(* CODESYS project Teste.project

Project tree, tasks and I/O mapping:
  Device : CODESYS Control Win V3, 3S - Smart Software Solutions GmbH, order no. 305021, version 3.5.11.40
    application Application
      libraries: Standard, * (System)
      task MainTask (cyclic, interval t#20ms, priority 1) calls Main
      program Main [ST]
      global variables Variaveis
      Carregamento/
        function UpdateAlarms [ST]
        function IniciarProcessoCarregamento [ST]
        function ExecutarCarregamento [ST]
        function ContinuarCarregamento [ST]
        function DesligarEquipamentosAposCarregamento [ST]
        function block ControleCarregamento [ST]
      ControleDescarregamento/
        function block ControleDescarregamento [ST]
        function UpdateAlarmsDescarregamento [ST]
        function IniciarProcessoDescarregamento [ST]
        function ExecutarDescarregamento [ST]
        function DesligarEquipamentosAposDescarregamento [ST]
      Geral/
        function VerificarCondicoesMudancaModo [ST]
      Symbols
*)

// Device/Application/Variaveis
VAR_GLOBAL
    // Variáveis de Comando
    CMD_INICIAR_CARREGAMENTO: BOOL := FALSE;
    CMD_INICIAR_DESCARREGAMENTO: BOOL := FALSE;

    // Variáveis do Caminhão
    CAMINHAO_POSICIONADO: BOOL := FALSE;
    CAPACIDADE_CAMINHAO: REAL := 0.0;

    // Variáveis dos Silos
    PESO_SILO1: REAL := 0.0;
    PESO_SILO2: REAL := 0.0;
    NIVEL_BAIXO_SILO1: BOOL := FALSE;
    NIVEL_BAIXO_SILO2: BOOL := FALSE;

    // Variáveis de Equipamentos
    VENTILACAO_SILO1: BOOL := FALSE;
    VENTILACAO_SILO2: BOOL := FALSE;
    ALIMENTADOR_MOEGA1_ON: BOOL := FALSE;
    ALIMENTADOR_MOEGA2_ON: BOOL := FALSE;
    TRANSPORTADOR_SAIDA_ON: BOOL := FALSE;
    MOEGA_PESAGEM_ON: BOOL := FALSE;
    TRANSPORTADOR_ENTRADA_ON: BOOL := FALSE;

    // Variáveis de Pesagem
    PESO_MOEGA: REAL := 0.0;
    TaxaTransferencia: REAL := 0.0;

    // Variáveis de Alarmes
    ALARME_CARREGAMENTO: BOOL := FALSE;
    ALARME_DESCARREGAMENTO: BOOL := FALSE;

    // Variáveis de Controle de Processo
    INICIAR_CARREGAMENTO: BOOL := FALSE;
    INICIAR_DESCARREGAMENTO: BOOL := FALSE;
    inicio_carregamento: TIME;
    inicio_descarregamento: TIME;
    SiloSelecionado: INT := 0;
	DESVIADOR_MANGUEIRA: INT;

    // Variáveis Adicionais
    VAGAO_POSICIONADO: BOOL := FALSE;
    CAPACIDADE_VAGAO: REAL := 1000.0; // Capacidade do vagão em kg

    // Modo de Operação: TRUE para Automático, FALSE para Manual
    Modo_Automatico_Carregamento: BOOL := FALSE; // FALSE = Manual, TRUE = Automático
    Modo_Automatico_Descarregamento: BOOL := FALSE; // FALSE = Manual, TRUE = Automático

    // Variáveis de Controle Manual
    CMD_MANUAL_VENTILACAO_SILO1: BOOL := FALSE;
    CMD_MANUAL_VENTILACAO_SILO2: BOOL := FALSE;
    CMD_MANUAL_ALIMENTADOR_MOEGA1_ON: BOOL := FALSE;
    CMD_MANUAL_ALIMENTADOR_MOEGA2_ON: BOOL := FALSE;
    CMD_MANUAL_TRANSPORTADOR_ENTRADA_ON: BOOL := FALSE;
    CMD_MANUAL_TRANSPORTADOR_SAIDA_ON: BOOL := FALSE;
    CMD_MANUAL_MOEGA_PESAGEM_ON: BOOL := FALSE;
    CMD_MANUAL_ALIMENTADOR_SAIDA_ON: BOOL := FALSE;

    // Condições de Equipamentos e Alarmes
    Equipamentos_Desligados: BOOL := TRUE;
    Alarmes_Ativos: BOOL := FALSE;
    Alarme_Nivel_Baixo_Ativo: BOOL := FALSE;
    Alarme_Nivel_Alto_Ativo: BOOL := FALSE;
END_VAR

// Device/Application/Main
PROGRAM Main
VAR_INPUT
    
    CMD_INICIAR_CARREGAMENTO: BOOL;
    CMD_INICIAR_DESCARREGAMENTO: BOOL;

    CAMINHAO_POSICIONADO: BOOL;
    CAPACIDADE_CAMINHAO: REAL;
    
    PESO_SILO1: REAL;
    PESO_SILO2: REAL;

    Modo_Automatico: BOOL; 

    CMD_MANUAL_VENTILACAO_SILO1: BOOL;
    CMD_MANUAL_VENTILACAO_SILO2: BOOL;
    CMD_MANUAL_ALIMENTADOR_MOEGA1_ON: BOOL;
    CMD_MANUAL_ALIMENTADOR_MOEGA2_ON: BOOL;
    CMD_MANUAL_TRANSPORTADOR_ENTRADA_ON: BOOL;
    CMD_MANUAL_TRANSPORTADOR_SAIDA_ON: BOOL;
    CMD_MANUAL_MOEGA_PESAGEM_ON: BOOL;
    CMD_MANUAL_ALIMENTADOR_SAIDA_ON: BOOL;
END_VAR

VAR_OUTPUT
    
    VENTILACAO_SILO1: BOOL;
    VENTILACAO_SILO2: BOOL;
    ALIMENTADOR_MOEGA1_ON: BOOL;
    ALIMENTADOR_MOEGA2_ON: BOOL;
    TRANSPORTADOR_SAIDA_ON: BOOL;
    MOEGA_PESAGEM_ON: BOOL;
    TRANSPORTADOR_ENTRADA_ON: BOOL;
    DESVIADOR_MANGUEIRA: INT;
END_VAR

VAR
    
    NIVEL_BAIXO_SILO1: BOOL;
    NIVEL_BAIXO_SILO2: BOOL;
    NIVEL_ALTO_SILO1: BOOL;
    NIVEL_ALTO_SILO2: BOOL;
    
    PESO_MOEGA: REAL;
    TaxaTransferenciaCarregamento: REAL := 50.0;
    TaxaTransferenciaDescarregamento: REAL := 100.0;
    
    ALARME_CARREGAMENTO: BOOL;
    ALARME_DESCARREGAMENTO: BOOL;
    
    INICIAR_CARREGAMENTO: BOOL;
    INICIAR_DESCARREGAMENTO: BOOL;
    inicio_carregamento: TIME;
    inicio_descarregamento: TIME;
    SiloSelecionado: INT;
    
    VAGAO_POSICIONADO: BOOL;
    CAPACIDADE_VAGAO: REAL := 1000.0;
    VAGAO_CAPACIDADE_RESTANTE: REAL := 0.0; 
    VAGAO_POSICIONADO_ANTERIOR: BOOL := FALSE;
    
    lastUpdateTime: TIME;
    elapsedTime: REAL;
    CAMINHAO_CHEIO: BOOL;
    equipmentOffTime: TIME;
    VAGAO_CHEIO: BOOL; 
END_VAR

//
// Update Alarms
//ALARME_CARREGAMENTO := NOT CAMINHAO_POSICIONADO OR (CAPACIDADE_CAMINHAO < 200 OR CAPACIDADE_CAMINHAO > 800);
//IF ALARME_CARREGAMENTO THEN
  //  INICIAR_CARREGAMENTO := FALSE;
//END_IF;

//ALARME_DESCARREGAMENTO := NOT VAGAO_POSICIONADO OR (PESO_SILO1 >= 2400 OR PESO_SILO2 >= 2400);
//IF ALARME_DESCARREGAMENTO THEN
  //  INICIAR_DESCARREGAMENTO := FALSE;
//END_IF;

IF PESO_SILO1 < 100 THEN
    NIVEL_BAIXO_SILO1 := TRUE;
ELSE
    NIVEL_BAIXO_SILO1 := FALSE;    
END_IF

IF PESO_SILO2 < 100 THEN
    NIVEL_BAIXO_SILO2 := TRUE;
ELSE
    NIVEL_BAIXO_SILO2 := FALSE;    
END_IF

IF PESO_SILO1 > 2400 THEN
	NIVEL_ALTO_SILO1 := TRUE;
ELSE
    NIVEL_ALTO_SILO1 := FALSE;	
END_IF

IF PESO_SILO2 > 2400 THEN
	NIVEL_ALTO_SILO2 := TRUE;
ELSE 
    NIVEL_ALTO_SILO2 := FALSE;	
END_IF

elapsedTime := TIME_TO_REAL(TIME() - lastUpdateTime) / 1000.0;
lastUpdateTime := TIME();

IF VAGAO_POSICIONADO AND NOT VAGAO_POSICIONADO_ANTERIOR THEN
    VAGAO_CAPACIDADE_RESTANTE := CAPACIDADE_VAGAO;
    VAGAO_POSICIONADO_ANTERIOR := TRUE;
	VAGAO_CHEIO := FALSE;
ELSIF NOT VAGAO_POSICIONADO THEN
    VAGAO_POSICIONADO_ANTERIOR := FALSE;
END_IF;


IF Modo_Automatico THEN
    
    IF NOT INICIAR_CARREGAMENTO AND CMD_INICIAR_CARREGAMENTO AND CAMINHAO_POSICIONADO AND ((PESO_SILO1 - 100) + (PESO_SILO2 - 100) >= CAPACIDADE_CAMINHAO) AND (CAPACIDADE_CAMINHAO >= 200 AND CAPACIDADE_CAMINHAO <= 800 AND (REAL_TO_INT(CAPACIDADE_CAMINHAO) MOD 50 = 0)) THEN
        INICIAR_CARREGAMENTO := TRUE;
        inicio_carregamento := TIME();
        ALARME_CARREGAMENTO := FALSE;

        
        IF PESO_SILO1 >= PESO_SILO2 THEN
            SiloSelecionado := 1;
            VENTILACAO_SILO1 := TRUE;
            ALIMENTADOR_MOEGA1_ON := TRUE;
            ALIMENTADOR_MOEGA2_ON := FALSE;
        ELSE
            SiloSelecionado := 2;
            VENTILACAO_SILO2 := TRUE;
            ALIMENTADOR_MOEGA2_ON := TRUE;
            ALIMENTADOR_MOEGA1_ON := FALSE;
        END_IF;
    END_IF;

    IF INICIAR_CARREGAMENTO THEN
        
        IF (PESO_SILO1 >= 100 OR PESO_SILO2 >= 100) THEN
            TRANSPORTADOR_SAIDA_ON := TRUE;
            MOEGA_PESAGEM_ON := TRUE;
           
            IF PESO_MOEGA <= CAPACIDADE_CAMINHAO  THEN
                PESO_MOEGA := PESO_MOEGA + TaxaTransferenciaCarregamento * elapsedTime;
                IF SiloSelecionado = 1 AND (NOT NIVEL_BAIXO_SILO1) THEN
                    PESO_SILO1 := PESO_SILO1 - TaxaTransferenciaCarregamento * elapsedTime;
					VENTILACAO_SILO1 := TRUE;
                    ALIMENTADOR_MOEGA1_ON := TRUE;
					VENTILACAO_SILO2 := FALSE;
                    ALIMENTADOR_MOEGA2_ON := FALSE;
                    IF NIVEL_BAIXO_SILO1 THEN
                        
                        SiloSelecionado := 2;
                        VENTILACAO_SILO1 := FALSE;
                        VENTILACAO_SILO2 := TRUE;
                        ALIMENTADOR_MOEGA1_ON := FALSE;
                        ALIMENTADOR_MOEGA2_ON := TRUE;
                    END_IF;
                ELSE
                    PESO_SILO2 := PESO_SILO2 - TaxaTransferenciaCarregamento * elapsedTime;
                    VENTILACAO_SILO2 := TRUE;
                    ALIMENTADOR_MOEGA2_ON := TRUE;
					VENTILACAO_SILO1 := FALSE;
                    ALIMENTADOR_MOEGA1_ON := FALSE;
                    IF NIVEL_BAIXO_SILO2 THEN
                        SiloSelecionado := 1;
                        VENTILACAO_SILO2 := FALSE;
                        VENTILACAO_SILO1 := TRUE;
                        ALIMENTADOR_MOEGA2_ON := FALSE;
                        ALIMENTADOR_MOEGA1_ON := TRUE;
                    END_IF;
                END_IF;
            END_IF
        ELSE
            ALARME_CARREGAMENTO := TRUE;
            INICIAR_CARREGAMENTO := FALSE;
        END_IF;

        IF PESO_MOEGA >= CAPACIDADE_CAMINHAO THEN
            CAMINHAO_CHEIO := TRUE;
            INICIAR_CARREGAMENTO := FALSE; 
            equipmentOffTime := TIME(); 
        END_IF;
    END_IF;

   
    IF CAMINHAO_CHEIO THEN
        IF (TIME() - equipmentOffTime >= T#1S) THEN
            MOEGA_PESAGEM_ON := FALSE;
        END_IF;
        IF (TIME() - equipmentOffTime >= T#2S) THEN
            TRANSPORTADOR_SAIDA_ON := FALSE;
        END_IF;
        IF (TIME() - equipmentOffTime >= T#3S) THEN
            ALIMENTADOR_MOEGA1_ON := FALSE;
            ALIMENTADOR_MOEGA2_ON := FALSE;
        END_IF;
        IF (TIME() - equipmentOffTime >= T#5S) THEN
            VENTILACAO_SILO1 := FALSE;
            VENTILACAO_SILO2 := FALSE;
            CAMINHAO_CHEIO := FALSE; 
        END_IF;
    END_IF;
	
    IF NOT INICIAR_DESCARREGAMENTO AND CMD_INICIAR_DESCARREGAMENTO AND VAGAO_POSICIONADO AND (PESO_SILO1 + PESO_SILO2 < 5000) AND (NOT VAGAO_CHEIO) AND NOT (NIVEL_ALTO_SILO1 AND NIVEL_ALTO_SILO2) THEN
        IF NOT ALARME_DESCARREGAMENTO THEN
            INICIAR_DESCARREGAMENTO := TRUE;
            inicio_descarregamento := TIME();
           
            IF (PESO_SILO1 <= PESO_SILO2) AND (NOT NIVEL_ALTO_SILO1) THEN
                //SiloSelecionado := 1;
                DESVIADOR_MANGUEIRA := 1;
                VENTILACAO_SILO1 := TRUE;
                VENTILACAO_SILO2 := FALSE;
            ELSE
               // SiloSelecionado := 2;
                DESVIADOR_MANGUEIRA := 2;
                VENTILACAO_SILO2 := TRUE;
                VENTILACAO_SILO1 := FALSE;
            END_IF;
        ELSE
            INICIAR_DESCARREGAMENTO := FALSE;
			ALARME_DESCARREGAMENTO  := TRUE;
        END_IF;
    END_IF;

    IF INICIAR_DESCARREGAMENTO THEN
        TRANSPORTADOR_ENTRADA_ON := TRUE;
        IF VAGAO_CAPACIDADE_RESTANTE > 0 THEN
            IF (NOT NIVEL_ALTO_SILO1) AND (DESVIADOR_MANGUEIRA = 1) THEN
                PESO_SILO1 := PESO_SILO1 + TaxaTransferenciaDescarregamento * elapsedTime;
                VAGAO_CAPACIDADE_RESTANTE := VAGAO_CAPACIDADE_RESTANTE - TaxaTransferenciaDescarregamento * elapsedTime;
				DESVIADOR_MANGUEIRA := 1;
				VENTILACAO_SILO1 := TRUE;
				VENTILACAO_SILO2 := FALSE;
                IF NIVEL_ALTO_SILO1 THEN
                    
                   //SiloSelecionado := 2;
                   DESVIADOR_MANGUEIRA := 2;
                   VENTILACAO_SILO1 := FALSE;
                   VENTILACAO_SILO2 := TRUE;
               END_IF;
            ELSE
                PESO_SILO2 := PESO_SILO2 + TaxaTransferenciaDescarregamento * elapsedTime;
                VAGAO_CAPACIDADE_RESTANTE := VAGAO_CAPACIDADE_RESTANTE - TaxaTransferenciaDescarregamento * elapsedTime;
				DESVIADOR_MANGUEIRA := 2;
				VENTILACAO_SILO2 := TRUE;
				VENTILACAO_SILO1 := FALSE;
                 IF NIVEL_ALTO_SILO2 THEN
                   
                   //SiloSelecionado := 1;
                   DESVIADOR_MANGUEIRA := 1;
                   VENTILACAO_SILO2 := FALSE;
                   VENTILACAO_SILO1 := TRUE;
                END_IF;
            END_IF;

            IF VAGAO_CAPACIDADE_RESTANTE <= 0 THEN
                VAGAO_CHEIO := TRUE;
                INICIAR_DESCARREGAMENTO := FALSE; 
                equipmentOffTime := TIME(); 
            END_IF;
        END_IF;
    END_IF;

    IF VAGAO_CHEIO THEN
        IF (TIME() - equipmentOffTime >= T#2S) THEN
            TRANSPORTADOR_ENTRADA_ON := FALSE;
        END_IF;
        IF (TIME() - equipmentOffTime >= T#5S) THEN
            IF DESVIADOR_MANGUEIRA = 1 THEN
                VENTILACAO_SILO1 := FALSE;
            ELSE
                VENTILACAO_SILO2 := FALSE;
            END_IF;
           // VAGAO_CHEIO := FALSE; 
        END_IF;
    END_IF;
END_IF


IF NOT Modo_Automatico THEN
    
    VENTILACAO_SILO1 := CMD_MANUAL_VENTILACAO_SILO1;
    VENTILACAO_SILO2 := CMD_MANUAL_VENTILACAO_SILO2;
    ALIMENTADOR_MOEGA1_ON := CMD_MANUAL_ALIMENTADOR_MOEGA1_ON;
    ALIMENTADOR_MOEGA2_ON := CMD_MANUAL_ALIMENTADOR_MOEGA2_ON;
    TRANSPORTADOR_SAIDA_ON := CMD_MANUAL_TRANSPORTADOR_SAIDA_ON;
    MOEGA_PESAGEM_ON := CMD_MANUAL_MOEGA_PESAGEM_ON;
    
    // Manual Unloading
    VENTILACAO_SILO1 := CMD_MANUAL_VENTILACAO_SILO1;
    VENTILACAO_SILO2 := CMD_MANUAL_VENTILACAO_SILO2;
    TRANSPORTADOR_ENTRADA_ON := CMD_MANUAL_TRANSPORTADOR_ENTRADA_ON;
END_IF;

END_PROGRAM

// Device/Application/Carregamento/UpdateAlarms
FUNCTION UpdateAlarms : BOOL
VAR_INPUT
    CAMINHAO_POSICIONADO: BOOL;
    CAPACIDADE_CAMINHAO: REAL;
END_VAR
VAR_OUTPUT
    ALARME_CARREGAMENTO: BOOL;
    INICIAR_CARREGAMENTO: BOOL;
END_VAR

ALARME_CARREGAMENTO := NOT CAMINHAO_POSICIONADO OR (CAPACIDADE_CAMINHAO < 200 OR CAPACIDADE_CAMINHAO > 800);
IF ALARME_CARREGAMENTO THEN
    INICIAR_CARREGAMENTO := FALSE;
END_IF;
UpdateAlarms := ALARME_CARREGAMENTO;

END_FUNCTION

// Device/Application/Carregamento/IniciarProcessoCarregamento
FUNCTION IniciarProcessoCarregamento : BOOL
VAR_INPUT
    CAMINHAO_POSICIONADO: BOOL;
    CAPACIDADE_CAMINHAO: REAL;
    PESO_SILO1: REAL;
    PESO_SILO2: REAL;
    ALARME_CARREGAMENTO: BOOL;
END_VAR
VAR_OUTPUT
    INICIAR_CARREGAMENTO: BOOL;
    inicio_carregamento: TIME;
END_VAR

IF CAMINHAO_POSICIONADO AND ((PESO_SILO1 - 100) + (PESO_SILO2 - 100) >= CAPACIDADE_CAMINHAO) THEN
    IF (CAPACIDADE_CAMINHAO >= 200 AND CAPACIDADE_CAMINHAO <= 800 AND (REAL_TO_INT(CAPACIDADE_CAMINHAO) MOD 50 = 0)) AND NOT ALARME_CARREGAMENTO THEN
        INICIAR_CARREGAMENTO := TRUE;
        inicio_carregamento := TIME();
        ALARME_CARREGAMENTO := FALSE; // Garante que o alarme de carregamento está resetado.
        IniciarProcessoCarregamento := TRUE;
    ELSE
        ALARME_CARREGAMENTO := TRUE;
        INICIAR_CARREGAMENTO := FALSE; // Não iniciar o carregamento se a capacidade não for adequada.
        IniciarProcessoCarregamento := FALSE;
    END_IF;
ELSE
    ALARME_CARREGAMENTO := TRUE;
    INICIAR_CARREGAMENTO := FALSE;
    IniciarProcessoCarregamento := FALSE;
END_IF;

END_FUNCTION

// Device/Application/Carregamento/ExecutarCarregamento
FUNCTION ExecutarCarregamento
VAR_INPUT
    INICIAR_CARREGAMENTO: BOOL;
    PESO_SILO1: REAL;
    PESO_SILO2: REAL;
    CAPACIDADE_CAMINHAO: REAL;
    ALARME_CARREGAMENTO: BOOL;
END_VAR
VAR_OUTPUT
    VENTILACAO_SILO1: BOOL;
    VENTILACAO_SILO2: BOOL;
    ALIMENTADOR_MOEGA1_ON: BOOL;
    ALIMENTADOR_MOEGA2_ON: BOOL;
    TRANSPORTADOR_SAIDA_ON: BOOL;
    MOEGA_PESAGEM_ON: BOOL;
END_VAR

IF INICIAR_CARREGAMENTO THEN
    IF (PESO_SILO1 + PESO_SILO2 >= CAPACIDADE_CAMINHAO) THEN
        IF (PESO_SILO1 >= PESO_SILO2 AND NOT NIVEL_BAIXO_SILO1) OR NIVEL_BAIXO_SILO2 THEN
            VENTILACAO_SILO1 := TRUE;
            ALIMENTADOR_MOEGA1_ON := TRUE;
            ALIMENTADOR_MOEGA2_ON := FALSE;
        ELSIF (PESO_SILO2 > PESO_SILO1 AND NOT NIVEL_BAIXO_SILO2) OR NIVEL_BAIXO_SILO1 THEN
            VENTILACAO_SILO2 := TRUE;
            ALIMENTADOR_MOEGA2_ON := TRUE;
            ALIMENTADOR_MOEGA1_ON := FALSE;
        END_IF;

        TRANSPORTADOR_SAIDA_ON := TRUE;
        MOEGA_PESAGEM_ON := TRUE;
        ContinuarCarregamento(ALIMENTADOR_MOEGA1_ON := ALIMENTADOR_MOEGA1_ON, ALIMENTADOR_MOEGA2_ON := ALIMENTADOR_MOEGA2_ON, TaxaTransferencia := TaxaTransferencia, PESO_SILO1 := PESO_SILO1, PESO_SILO2 := PESO_SILO2, CAPACIDADE_CAMINHAO := CAPACIDADE_CAMINHAO, NIVEL_BAIXO_SILO1 := NIVEL_BAIXO_SILO1, NIVEL_BAIXO_SILO2 := NIVEL_BAIXO_SILO2, PESO_MOEGA => PESO_MOEGA);
    ELSE
        ALARME_CARREGAMENTO := TRUE;
        INICIAR_CARREGAMENTO := FALSE;
    END_IF;
END_IF;

END_FUNCTION

// Device/Application/Carregamento/ContinuarCarregamento
FUNCTION ContinuarCarregamento
VAR_INPUT
    ALIMENTADOR_MOEGA1_ON: BOOL;
    ALIMENTADOR_MOEGA2_ON: BOOL;
    TaxaTransferencia: REAL;
    PESO_SILO1: REAL;
    PESO_SILO2: REAL;
    CAPACIDADE_CAMINHAO: REAL;
    NIVEL_BAIXO_SILO1: BOOL;
    NIVEL_BAIXO_SILO2: BOOL;
END_VAR
VAR_OUTPUT
    PESO_MOEGA: REAL;
END_VAR

IF ALIMENTADOR_MOEGA1_ON THEN
    PESO_SILO1 := PESO_SILO1 - TaxaTransferencia;
END_IF;
IF ALIMENTADOR_MOEGA2_ON THEN
    PESO_SILO2 := PESO_SILO2 - TaxaTransferencia;
END_IF;
PESO_MOEGA := PESO_MOEGA + TaxaTransferencia;

IF PESO_MOEGA >= CAPACIDADE_CAMINHAO OR (NIVEL_BAIXO_SILO1 AND ALIMENTADOR_MOEGA1_ON) OR (NIVEL_BAIXO_SILO2 AND ALIMENTADOR_MOEGA2_ON) THEN
    DesligarEquipamentosAposCarregamento(inicio_carregamento, MOEGA_PESAGEM_ON, TRANSPORTADOR_SAIDA_ON, ALIMENTADOR_MOEGA1_ON, ALIMENTADOR_MOEGA2_ON, VENTILACAO_SILO1, VENTILACAO_SILO2, INICIAR_CARREGAMENTO);
END_IF;

END_FUNCTION

// Device/Application/Carregamento/DesligarEquipamentosAposCarregamento
FUNCTION DesligarEquipamentosAposCarregamento
VAR_INPUT
    inicio_carregamento: TIME;
    MOEGA_PESAGEM_ON: BOOL;
    TRANSPORTADOR_SAIDA_ON: BOOL;
    ALIMENTADOR_MOEGA1_ON: BOOL;
    ALIMENTADOR_MOEGA2_ON: BOOL;
    VENTILACAO_SILO1: BOOL;
    VENTILACAO_SILO2: BOOL;
    INICIAR_CARREGAMENTO: BOOL;
END_VAR

IF (TIME() - inicio_carregamento >= T#1S) AND MOEGA_PESAGEM_ON THEN
    MOEGA_PESAGEM_ON := FALSE; // Desliga a moega de pesagem após 1 segundo do término do carregamento
END_IF;

IF (TIME() - inicio_carregamento >= T#2S) AND TRANSPORTADOR_SAIDA_ON THEN
    TRANSPORTADOR_SAIDA_ON := FALSE; // Desliga o transportador de saída após 2 segundos
END_IF;

IF (TIME() - inicio_carregamento >= T#3S) AND (ALIMENTADOR_MOEGA1_ON OR ALIMENTADOR_MOEGA2_ON) THEN
    ALIMENTADOR_MOEGA1_ON := FALSE; // Desliga o alimentador da moega 1 após 3 segundos
    ALIMENTADOR_MOEGA2_ON := FALSE; // Desliga o alimentador da moega 2 após 3 segundos
END_IF;

IF (TIME() - inicio_carregamento >= T#5S) THEN
    VENTILACAO_SILO1 := FALSE; // Desliga a ventilação do Silo 1 após 5 segundos
    VENTILACAO_SILO2 := FALSE; // Desliga a ventilação do Silo 2 após 5 segundos
    INICIAR_CARREGAMENTO := FALSE; // Sinaliza que o processo de carregamento está completamente finalizado
END_IF;

END_FUNCTION

// Device/Application/Carregamento/ControleCarregamento
FUNCTION_BLOCK ControleCarregamento
VAR_INPUT
    CMD_INICIAR_CARREGAMENTO: BOOL;
    CAMINHAO_POSICIONADO: BOOL;
    CAPACIDADE_CAMINHAO: REAL;
    PESO_SILO1: REAL;
    PESO_SILO2: REAL;
    TaxaTransferencia: REAL;
    // Variáveis de Comando Manual
    CMD_MANUAL_VENTILACAO_SILO1: BOOL;
    CMD_MANUAL_VENTILACAO_SILO2: BOOL;
    CMD_MANUAL_ALIMENTADOR_MOEGA1_ON: BOOL;
    CMD_MANUAL_ALIMENTADOR_MOEGA2_ON: BOOL;
    CMD_MANUAL_TRANSPORTADOR_SAIDA_ON: BOOL;
    CMD_MANUAL_MOEGA_PESAGEM_ON: BOOL;
END_VAR
VAR_OUTPUT
    INICIAR_CARREGAMENTO: BOOL;
    VENTILACAO_SILO1: BOOL;
    VENTILACAO_SILO2: BOOL;
    ALIMENTADOR_MOEGA1_ON: BOOL;
    ALIMENTADOR_MOEGA2_ON: BOOL;
    TRANSPORTADOR_SAIDA_ON: BOOL;
    MOEGA_PESAGEM_ON: BOOL;
    ALARME_CARREGAMENTO: BOOL;
END_VAR
VAR
    inicio_carregamento: TIME;
    PESO_MOEGA: REAL;
END_VAR

IF VerificarCondicoesMudancaModo() THEN
    Modo_Automatico_Carregamento := Modo_Automatico_Carregamento;
END_IF;

IF Modo_Automatico_Carregamento THEN
    // Lógica para modo automático
    ALARME_CARREGAMENTO := UpdateAlarms(CAMINHAO_POSICIONADO := CAMINHAO_POSICIONADO, CAPACIDADE_CAMINHAO := CAPACIDADE_CAMINHAO, INICIAR_CARREGAMENTO => INICIAR_CARREGAMENTO);

    IF CMD_INICIAR_CARREGAMENTO THEN
        IF IniciarProcessoCarregamento(CAMINHAO_POSICIONADO := CAMINHAO_POSICIONADO, CAPACIDADE_CAMINHAO := CAPACIDADE_CAMINHAO, PESO_SILO1 := PESO_SILO1, PESO_SILO2 := PESO_SILO2, ALARME_CARREGAMENTO := ALARME_CARREGAMENTO, INICIAR_CARREGAMENTO => INICIAR_CARREGAMENTO, inicio_carregamento => inicio_carregamento) THEN
            ExecutarCarregamento(INICIAR_CARREGAMENTO := INICIAR_CARREGAMENTO, PESO_SILO1 := PESO_SILO1, PESO_SILO2 := PESO_SILO2, CAPACIDADE_CAMINHAO := CAPACIDADE_CAMINHAO, ALARME_CARREGAMENTO := ALARME_CARREGAMENTO, VENTILACAO_SILO1 => VENTILACAO_SILO1, VENTILACAO_SILO2 => VENTILACAO_SILO2, ALIMENTADOR_MOEGA1_ON => ALIMENTADOR_MOEGA1_ON, ALIMENTADOR_MOEGA2_ON => ALIMENTADOR_MOEGA2_ON, TRANSPORTADOR_SAIDA_ON => TRANSPORTADOR_SAIDA_ON, MOEGA_PESAGEM_ON => MOEGA_PESAGEM_ON);
        END_IF;
    END_IF;

    DesligarEquipamentosAposCarregamento(inicio_carregamento := inicio_carregamento, MOEGA_PESAGEM_ON := MOEGA_PESAGEM_ON, TRANSPORTADOR_SAIDA_ON := TRANSPORTADOR_SAIDA_ON, ALIMENTADOR_MOEGA1_ON := ALIMENTADOR_MOEGA1_ON, ALIMENTADOR_MOEGA2_ON := ALIMENTADOR_MOEGA2_ON, VENTILACAO_SILO1 := VENTILACAO_SILO1, VENTILACAO_SILO2 := VENTILACAO_SILO2, INICIAR_CARREGAMENTO := INICIAR_CARREGAMENTO);
ELSE
    // Lógica para modo manual
    VENTILACAO_SILO1 := CMD_MANUAL_VENTILACAO_SILO1;
    VENTILACAO_SILO2 := CMD_MANUAL_VENTILACAO_SILO2;
    ALIMENTADOR_MOEGA1_ON := CMD_MANUAL_ALIMENTADOR_MOEGA1_ON;
    ALIMENTADOR_MOEGA2_ON := CMD_MANUAL_ALIMENTADOR_MOEGA2_ON;
    TRANSPORTADOR_SAIDA_ON := CMD_MANUAL_TRANSPORTADOR_SAIDA_ON;
    MOEGA_PESAGEM_ON := CMD_MANUAL_MOEGA_PESAGEM_ON;
END_IF;

END_FUNCTION_BLOCK

// Device/Application/Geral/VerificarCondicoesMudancaModo
FUNCTION VerificarCondicoesMudancaModo : BOOL
VAR_OUTPUT
    Equipamentos_Desligados: BOOL;
    Alarmes_Ativos: BOOL;
    Alarme_Nivel_Baixo_Ativo: BOOL;
    Alarme_Nivel_Alto_Ativo: BOOL;
END_VAR

Equipamentos_Desligados := NOT (ALIMENTADOR_MOEGA1_ON OR ALIMENTADOR_MOEGA2_ON OR TRANSPORTADOR_ENTRADA_ON OR TRANSPORTADOR_SAIDA_ON OR VENTILACAO_SILO1 OR VENTILACAO_SILO2 OR MOEGA_PESAGEM_ON);

// Verifica se há alarmes ativos (exceto os alarmes de nível baixo e alto)
Alarmes_Ativos := ALARME_CARREGAMENTO OR ALARME_DESCARREGAMENTO;

// Verifica se há alarmes de nível baixo ou alto ativos
Alarme_Nivel_Baixo_Ativo := NIVEL_BAIXO_SILO1 OR NIVEL_BAIXO_SILO2;
Alarme_Nivel_Alto_Ativo := PESO_SILO1 > 2400 OR PESO_SILO2 > 2400;

// Retorna TRUE se todos os equipamentos estiverem desligados e não houver alarmes ativos, exceto os de nível baixo e alto
VerificarCondicoesMudancaModo := Equipamentos_Desligados AND NOT Alarmes_Ativos;

END_FUNCTION

// Device/Application/ControleDescarregamento/ControleDescarregamento
FUNCTION_BLOCK ControleDescarregamento
VAR_INPUT
    CMD_INICIAR_DESCARREGAMENTO: BOOL;
    VAGAO_POSICIONADO: BOOL;
    PESO_SILO1: REAL;
    PESO_SILO2: REAL;
    TaxaTransferencia: REAL;
    // Variáveis de Comando Manual
    CMD_MANUAL_VENTILACAO_SILO1: BOOL;
    CMD_MANUAL_VENTILACAO_SILO2: BOOL;
    CMD_MANUAL_TRANSPORTADOR_ENTRADA_ON: BOOL;
END_VAR
VAR_OUTPUT
    INICIAR_DESCARREGAMENTO: BOOL;
    VENTILACAO_SILO1: BOOL;
    VENTILACAO_SILO2: BOOL;
    TRANSPORTADOR_ENTRADA_ON: BOOL;
    ALARME_DESCARREGAMENTO: BOOL;
END_VAR
VAR
    inicio_descarregamento: TIME;
    SiloSelecionado: INT;
    CAPACIDADE_VAGAO: REAL := 1000.0; // Capacidade do vagão em kg
END_VAR

IF VerificarCondicoesMudancaModo() THEN
    Modo_Automatico_Descarregamento := Modo_Automatico_Descarregamento;
END_IF;

IF Modo_Automatico_Descarregamento THEN
    // Lógica para modo automático
    ALARME_DESCARREGAMENTO := UpdateAlarmsDescarregamento(VAGAO_POSICIONADO := VAGAO_POSICIONADO, PESO_SILO1 := PESO_SILO1, PESO_SILO2 := PESO_SILO2, INICIAR_DESCARREGAMENTO => INICIAR_DESCARREGAMENTO);

    IF CMD_INICIAR_DESCARREGAMENTO THEN
        IF IniciarProcessoDescarregamento(VAGAO_POSICIONADO := VAGAO_POSICIONADO, PESO_SILO1 := PESO_SILO1, PESO_SILO2 := PESO_SILO2, ALARME_DESCARREGAMENTO := ALARME_DESCARREGAMENTO, INICIAR_DESCARREGAMENTO => INICIAR_DESCARREGAMENTO, inicio_descarregamento => inicio_descarregamento, SiloSelecionado => SiloSelecionado, VENTILACAO_SILO1 => VENTILACAO_SILO1, VENTILACAO_SILO2 => VENTILACAO_SILO2) THEN
            ExecutarDescarregamento(INICIAR_DESCARREGAMENTO := INICIAR_DESCARREGAMENTO, PESO_SILO1 := PESO_SILO1, PESO_SILO2 := PESO_SILO2, inicio_descarregamento := inicio_descarregamento, SiloSelecionado := SiloSelecionado, CAPACIDADE_VAGAO := CAPACIDADE_VAGAO, VENTILACAO_SILO1 => VENTILACAO_SILO1, VENTILACAO_SILO2 => VENTILACAO_SILO2, TRANSPORTADOR_ENTRADA_ON => TRANSPORTADOR_ENTRADA_ON);
        END_IF;
    END_IF;

    DesligarEquipamentosAposDescarregamento(inicio_descarregamento := inicio_descarregamento, SiloSelecionado := SiloSelecionado, TRANSPORTADOR_ENTRADA_ON := TRANSPORTADOR_ENTRADA_ON, VENTILACAO_SILO1 := VENTILACAO_SILO1, VENTILACAO_SILO2 := VENTILACAO_SILO2, INICIAR_DESCARREGAMENTO := INICIAR_DESCARREGAMENTO);
ELSE
    // Lógica para modo manual
    VENTILACAO_SILO1 := CMD_MANUAL_VENTILACAO_SILO1;
    VENTILACAO_SILO2 := CMD_MANUAL_VENTILACAO_SILO2;
    TRANSPORTADOR_ENTRADA_ON := CMD_MANUAL_TRANSPORTADOR_ENTRADA_ON;
END_IF;

END_FUNCTION_BLOCK

// Device/Application/ControleDescarregamento/UpdateAlarmsDescarregamento
FUNCTION UpdateAlarmsDescarregamento : BOOL
VAR_INPUT
    VAGAO_POSICIONADO: BOOL;
    PESO_SILO1: REAL;
    PESO_SILO2: REAL;
END_VAR
VAR_OUTPUT
    ALARME_DESCARREGAMENTO: BOOL;
    INICIAR_DESCARREGAMENTO: BOOL;
END_VAR


ALARME_DESCARREGAMENTO := NOT VAGAO_POSICIONADO OR (PESO_SILO1 >= 2400 OR PESO_SILO2 >= 2400);
IF ALARME_DESCARREGAMENTO THEN
    INICIAR_DESCARREGAMENTO := FALSE;
END_IF;
UpdateAlarmsDescarregamento := ALARME_DESCARREGAMENTO;

END_FUNCTION

// Device/Application/ControleDescarregamento/IniciarProcessoDescarregamento
FUNCTION IniciarProcessoDescarregamento : BOOL
VAR_INPUT
    VAGAO_POSICIONADO: BOOL;
    PESO_SILO1: REAL;
    PESO_SILO2: REAL;
    ALARME_DESCARREGAMENTO: BOOL;
END_VAR
VAR_OUTPUT
    INICIAR_DESCARREGAMENTO: BOOL;
    inicio_descarregamento: TIME;
    SiloSelecionado: INT;
    VENTILACAO_SILO1: BOOL;
    VENTILACAO_SILO2: BOOL;
END_VAR

IF VAGAO_POSICIONADO AND (PESO_SILO1 + PESO_SILO2 < 5000) THEN
    IF NOT ALARME_DESCARREGAMENTO THEN
        INICIAR_DESCARREGAMENTO := TRUE;
        inicio_descarregamento := TIME();
        
        // Seleciona o silo para descarregamento
        IF PESO_SILO1 < PESO_SILO2 THEN
            SiloSelecionado := 1;
            VENTILACAO_SILO1 := TRUE;
        ELSE
            SiloSelecionado := 2;
            VENTILACAO_SILO2 := TRUE;
        END_IF;
        
        IniciarProcessoDescarregamento := TRUE; // O processo de descarregamento começará
    ELSE
        IniciarProcessoDescarregamento := FALSE; // O processo de descarregamento não começará
    END_IF;
ELSE
    ALARME_DESCARREGAMENTO := TRUE;
    IniciarProcessoDescarregamento := FALSE;
END_IF;

END_FUNCTION

// Device/Application/ControleDescarregamento/ExecutarDescarregamento
FUNCTION ExecutarDescarregamento
VAR_INPUT
    INICIAR_DESCARREGAMENTO: BOOL;
    PESO_SILO1: REAL;
    PESO_SILO2: REAL;
    inicio_descarregamento: TIME;
    SiloSelecionado: INT;
    CAPACIDADE_VAGAO: REAL;
END_VAR
VAR_OUTPUT
    VENTILACAO_SILO1: BOOL;
    VENTILACAO_SILO2: BOOL;
    TRANSPORTADOR_ENTRADA_ON: BOOL;
END_VAR
VAR
    tempo_atual: TIME;
    delta_tempo: UDINT;
END_VAR

IF INICIAR_DESCARREGAMENTO THEN
    TRANSPORTADOR_ENTRADA_ON := TRUE;
    tempo_atual := TIME();
    delta_tempo := TO_UDINT(tempo_atual - inicio_descarregamento); // Converte TIME para UDINT (milissegundos)
    
    IF SiloSelecionado = 1 THEN
        // Transfere grãos para o Silo 1
        PESO_SILO1 := PESO_SILO1 + 100 * (TO_REAL(delta_tempo) / 1000.0); // Converte milissegundos para segundos
        IF PESO_SILO1 >= 2400 THEN
            SiloSelecionado := 2;
            VENTILACAO_SILO1 := FALSE;
            VENTILACAO_SILO2 := TRUE;
        END_IF;
    ELSE
        // Transfere grãos para o Silo 2
        PESO_SILO2 := PESO_SILO2 + 100 * (TO_REAL(delta_tempo) / 1000.0); // Converte milissegundos para segundos
        IF PESO_SILO2 >= 2400 THEN
            SiloSelecionado := 1;
            VENTILACAO_SILO2 := FALSE;
            VENTILACAO_SILO1 := TRUE;
        END_IF;
    END_IF;
    
    // Verifica se o transportador está vazio
    IF PESO_SILO1 + PESO_SILO2 >= CAPACIDADE_VAGAO THEN
        DesligarEquipamentosAposDescarregamento(inicio_descarregamento, SiloSelecionado, TRANSPORTADOR_ENTRADA_ON, VENTILACAO_SILO1, VENTILACAO_SILO2, INICIAR_DESCARREGAMENTO);
    END_IF;
END_IF;

END_FUNCTION

// Device/Application/ControleDescarregamento/DesligarEquipamentosAposDescarregamento
FUNCTION DesligarEquipamentosAposDescarregamento
VAR_INPUT
    inicio_descarregamento: TIME;
    SiloSelecionado: INT;
    TRANSPORTADOR_ENTRADA_ON: BOOL;
    VENTILACAO_SILO1: BOOL;
    VENTILACAO_SILO2: BOOL;
    INICIAR_DESCARREGAMENTO: BOOL;
END_VAR

IF (TIME() - inicio_descarregamento >= T#2S) THEN
    TRANSPORTADOR_ENTRADA_ON := FALSE;
END_IF;

IF (TIME() - inicio_descarregamento >= T#5S) THEN
    IF SiloSelecionado = 1 THEN
        VENTILACAO_SILO1 := FALSE;
    ELSE
        VENTILACAO_SILO2 := FALSE;
    END_IF;
    INICIAR_DESCARREGAMENTO := FALSE; // Finaliza completamente o processo de descarregamento
END_IF;

END_FUNCTION
